(* CODESYS project WagoLibVisuIndustrialElements.library
   Description: Visualization objects for use with e!Cockpit programming environment
   Version: 1.0.0
   Title: WagoLibIndustrialVisuElements
   Author: JCox
   CompiledLibraryCompatibilityVersion: CODESYS V3.5 SP16 Patch 2
   Company: WAGO Corp. USA

Project tree, tasks and I/O mapping:
  libraries: VisuSymbols, 3.5.17.0 (System); WagoVisuIcons, 1.1.0.4 (WAGO)
  5ce3da45-db07-42e7-a21c-a00fff4ed8f6|Z:\Dropbox\Demos\Image Library\JPG Exports\blower1.png
  text list GlobalTextList
  5ce3da45-db07-42e7-a21c-a00fff4ed8f6|Z:\Dropbox\Demos\Image Library\JPG Exports\barrelblue.png
  visualisation GateValve1
  visualisation GlobeValve1
  visualisation Motor1
  visualisation Motor2
  visualisation Pump1
  visualisation Pump2
  visualisation Pump3
  visualisation Pump4
  visualisation Tank1
  visualisation Tank2
  visualisation Tank3
  visualisation Tank4
  visualisation Valve1
  visualisation Valve2
  image pool ImagePool
  5ce3da45-db07-42e7-a21c-a00fff4ed8f6|Z:\Dropbox\Demos\Image Library\JPG Exports\boiler1.png
  5ce3da45-db07-42e7-a21c-a00fff4ed8f6|Z:\Dropbox\Demos\Image Library\JPG Exports\barrelred.png
  visualisation Burner1
  5ce3da45-db07-42e7-a21c-a00fff4ed8f6|Z:\Dropbox\Demos\Image Library\JPG Exports\heatpipeOFF.png
  5ce3da45-db07-42e7-a21c-a00fff4ed8f6|Z:\Dropbox\Demos\Image Library\JPG Exports\heatpipeON.png
  5ce3da45-db07-42e7-a21c-a00fff4ed8f6|Z:\Dropbox\Demos\Image Library\JPG Exports\boiler2.png
  5ce3da45-db07-42e7-a21c-a00fff4ed8f6|Z:\Dropbox\Demos\Image Library\JPG Exports\box1.png
  5ce3da45-db07-42e7-a21c-a00fff4ed8f6|Z:\Dropbox\Demos\Image Library\JPG Exports\box2.png
  5ce3da45-db07-42e7-a21c-a00fff4ed8f6|Z:\Dropbox\Demos\Image Library\JPG Exports\check valveGRN.png
  5ce3da45-db07-42e7-a21c-a00fff4ed8f6|Z:\Dropbox\Demos\Image Library\JPG Exports\check valveGRN2.png
  5ce3da45-db07-42e7-a21c-a00fff4ed8f6|Z:\Dropbox\Demos\Image Library\JPG Exports\check valveGRY.png
  5ce3da45-db07-42e7-a21c-a00fff4ed8f6|Z:\Dropbox\Demos\Image Library\JPG Exports\check valveGRY2.png
  5ce3da45-db07-42e7-a21c-a00fff4ed8f6|Z:\Dropbox\Demos\Image Library\JPG Exports\check valveRED.png
  5ce3da45-db07-42e7-a21c-a00fff4ed8f6|Z:\Dropbox\Demos\Image Library\JPG Exports\check valveRED2.png
  5ce3da45-db07-42e7-a21c-a00fff4ed8f6|Z:\Dropbox\Demos\Image Library\JPG Exports\conveyor1.png
  5ce3da45-db07-42e7-a21c-a00fff4ed8f6|Z:\Dropbox\Demos\Image Library\JPG Exports\conveyor3.png
  5ce3da45-db07-42e7-a21c-a00fff4ed8f6|Z:\Dropbox\Demos\Image Library\JPG Exports\fireEMPTY.png
  5ce3da45-db07-42e7-a21c-a00fff4ed8f6|Z:\Dropbox\Demos\Image Library\JPG Exports\fireFULL.png
  5ce3da45-db07-42e7-a21c-a00fff4ed8f6|Z:\Dropbox\Demos\Image Library\JPG Exports\gatevalveGRN.png
  5ce3da45-db07-42e7-a21c-a00fff4ed8f6|Z:\Dropbox\Demos\Image Library\JPG Exports\gatevalveGRY.png
  5ce3da45-db07-42e7-a21c-a00fff4ed8f6|Z:\Dropbox\Demos\Image Library\JPG Exports\globevalveGRN.png
  5ce3da45-db07-42e7-a21c-a00fff4ed8f6|Z:\Dropbox\Demos\Image Library\JPG Exports\globevalveGRY.png
  5ce3da45-db07-42e7-a21c-a00fff4ed8f6|Z:\Dropbox\Demos\Image Library\JPG Exports\mixer1GRN.png
  5ce3da45-db07-42e7-a21c-a00fff4ed8f6|Z:\Dropbox\Demos\Image Library\JPG Exports\mixer1RED.png
  5ce3da45-db07-42e7-a21c-a00fff4ed8f6|Z:\Dropbox\Demos\Image Library\JPG Exports\motor1.png
  5ce3da45-db07-42e7-a21c-a00fff4ed8f6|Z:\Dropbox\Demos\Image Library\JPG Exports\motor1GRN.png
  5ce3da45-db07-42e7-a21c-a00fff4ed8f6|Z:\Dropbox\Demos\Image Library\JPG Exports\motor1RED.png
  5ce3da45-db07-42e7-a21c-a00fff4ed8f6|Z:\Dropbox\Demos\Image Library\JPG Exports\motorBLU1.png
  5ce3da45-db07-42e7-a21c-a00fff4ed8f6|Z:\Dropbox\Demos\Image Library\JPG Exports\motorBLU2.png
  5ce3da45-db07-42e7-a21c-a00fff4ed8f6|Z:\Dropbox\Demos\Image Library\JPG Exports\motorBLU3.png
  5ce3da45-db07-42e7-a21c-a00fff4ed8f6|Z:\Dropbox\Demos\Image Library\JPG Exports\motorGRN1.png
  5ce3da45-db07-42e7-a21c-a00fff4ed8f6|Z:\Dropbox\Demos\Image Library\JPG Exports\motorGRN2.png
  5ce3da45-db07-42e7-a21c-a00fff4ed8f6|Z:\Dropbox\Demos\Image Library\JPG Exports\motorGRN3.png
  5ce3da45-db07-42e7-a21c-a00fff4ed8f6|Z:\Dropbox\Demos\Image Library\JPG Exports\motorRED1.png
  5ce3da45-db07-42e7-a21c-a00fff4ed8f6|Z:\Dropbox\Demos\Image Library\JPG Exports\motorRED2.png
  5ce3da45-db07-42e7-a21c-a00fff4ed8f6|Z:\Dropbox\Demos\Image Library\JPG Exports\motorRED3.png
  5ce3da45-db07-42e7-a21c-a00fff4ed8f6|Z:\Dropbox\Demos\Image Library\JPG Exports\pipe1H.png
  5ce3da45-db07-42e7-a21c-a00fff4ed8f6|Z:\Dropbox\Demos\Image Library\JPG Exports\pipe1V.png
  5ce3da45-db07-42e7-a21c-a00fff4ed8f6|Z:\Dropbox\Demos\Image Library\JPG Exports\pipeJ1.png
  5ce3da45-db07-42e7-a21c-a00fff4ed8f6|Z:\Dropbox\Demos\Image Library\JPG Exports\pipeJ2.png
  5ce3da45-db07-42e7-a21c-a00fff4ed8f6|Z:\Dropbox\Demos\Image Library\JPG Exports\pipeJ3.png
  5ce3da45-db07-42e7-a21c-a00fff4ed8f6|Z:\Dropbox\Demos\Image Library\JPG Exports\pipeJ4.png
  5ce3da45-db07-42e7-a21c-a00fff4ed8f6|Z:\Dropbox\Demos\Image Library\JPG Exports\pipeT1.png
  5ce3da45-db07-42e7-a21c-a00fff4ed8f6|Z:\Dropbox\Demos\Image Library\JPG Exports\pipeT2.png
  5ce3da45-db07-42e7-a21c-a00fff4ed8f6|Z:\Dropbox\Demos\Image Library\JPG Exports\pipeT3.png
  5ce3da45-db07-42e7-a21c-a00fff4ed8f6|Z:\Dropbox\Demos\Image Library\JPG Exports\pipeT4.png
  5ce3da45-db07-42e7-a21c-a00fff4ed8f6|Z:\Dropbox\Demos\Image Library\JPG Exports\pipeX.png
  5ce3da45-db07-42e7-a21c-a00fff4ed8f6|Z:\Dropbox\Demos\Image Library\JPG Exports\pump1.png
  5ce3da45-db07-42e7-a21c-a00fff4ed8f6|Z:\Dropbox\Demos\Image Library\JPG Exports\pump2.png
  5ce3da45-db07-42e7-a21c-a00fff4ed8f6|Z:\Dropbox\Demos\Image Library\JPG Exports\pump3.png
  5ce3da45-db07-42e7-a21c-a00fff4ed8f6|Z:\Dropbox\Demos\Image Library\JPG Exports\pump4.png
  5ce3da45-db07-42e7-a21c-a00fff4ed8f6|Z:\Dropbox\Demos\Image Library\JPG Exports\tank2.png
  5ce3da45-db07-42e7-a21c-a00fff4ed8f6|Z:\Dropbox\Demos\Image Library\JPG Exports\tank1.png
  5ce3da45-db07-42e7-a21c-a00fff4ed8f6|Z:\Dropbox\Demos\Image Library\JPG Exports\tank3.png
  5ce3da45-db07-42e7-a21c-a00fff4ed8f6|Z:\Dropbox\Demos\Image Library\JPG Exports\tank4.png
  5ce3da45-db07-42e7-a21c-a00fff4ed8f6|Z:\Dropbox\Demos\Image Library\JPG Exports\tank5.png
  5ce3da45-db07-42e7-a21c-a00fff4ed8f6|Z:\Dropbox\Demos\Image Library\JPG Exports\tank6.png
  5ce3da45-db07-42e7-a21c-a00fff4ed8f6|Z:\Dropbox\Demos\Image Library\JPG Exports\tank7.png
*)

// /GateValve1
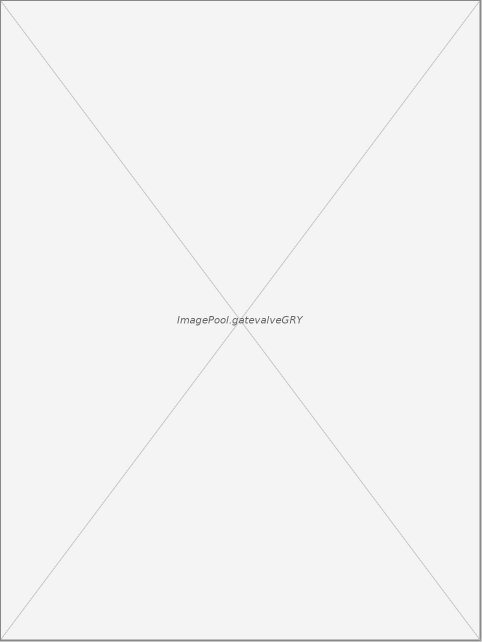
VISUALIZATION GateValve1  // 482x642
VAR_IN_OUT
	xOn		: BOOL;
END_VAR
    Image (0,0 480x640), invisible if: NOT xOn, image: ImagePool.gatevalveGRN
    Image (0,0 480x640), invisible if: xOn, image: ImagePool.gatevalveGRY
END_VISUALIZATION

// /GlobeValve1
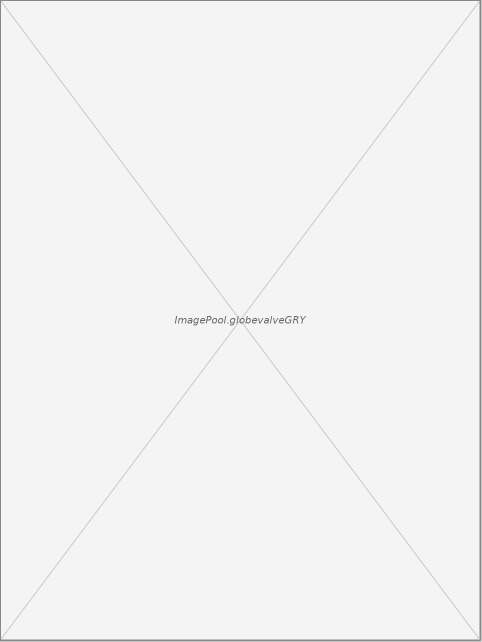
VISUALIZATION GlobeValve1  // 482x642
VAR_IN_OUT
	xOn		: BOOL;
END_VAR
    Image (0,0 480x640), invisible if: NOT xOn, image: ImagePool.globevalveGRN
    Image (0,0 480x640), invisible if: xOn, image: ImagePool.globevalveGRY
END_VISUALIZATION

// /Motor1
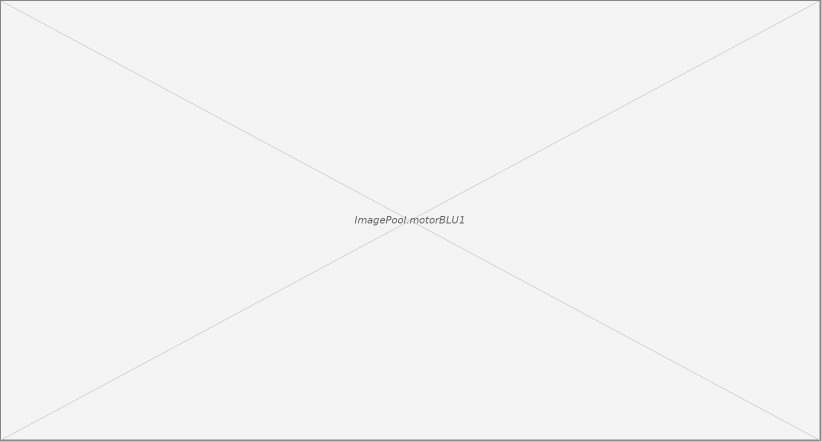
VISUALIZATION Motor1  // 822x442
VAR_IN_OUT
	xOn	: BOOL;
END_VAR
    Image (0,0 820x440), invisible if: NOT xOn, image: ImagePool.motorGRN1
    Image (0,0 820x440), invisible if: xOn, image: ImagePool.motorBLU1
END_VISUALIZATION

// /Motor2
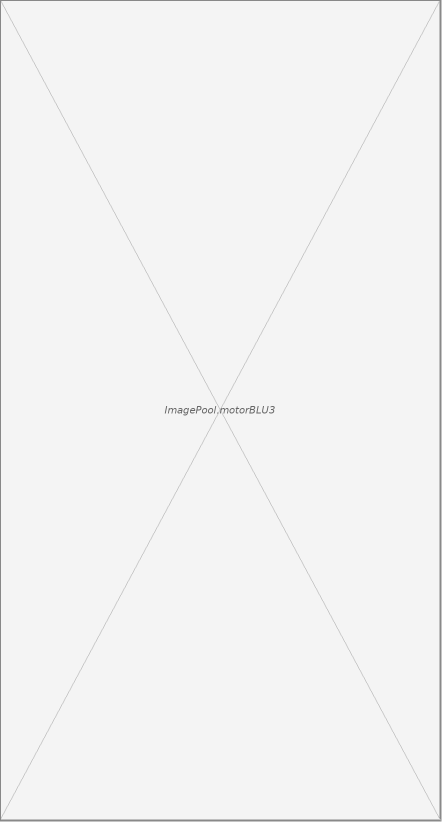
VISUALIZATION Motor2  // 442x822
VAR_IN_OUT
	xOn	: BOOL;
END_VAR
    Image (0,0 440x820), invisible if: NOT xOn, image: ImagePool.motorGRN3
    Image (0,0 440x820), invisible if: xOn, image: ImagePool.motorBLU3
END_VISUALIZATION

// /Pump1
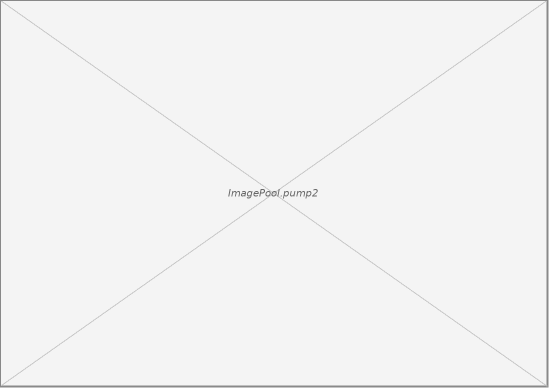
VISUALIZATION Pump1  // 549x388
VAR_IN_OUT
	xGo	: BOOL;
END_VAR
    Ellipse (125,44 300x300), colour toggle: xGo
    Image (0,0 547x386), image: ImagePool.pump2
END_VISUALIZATION

// /Pump2
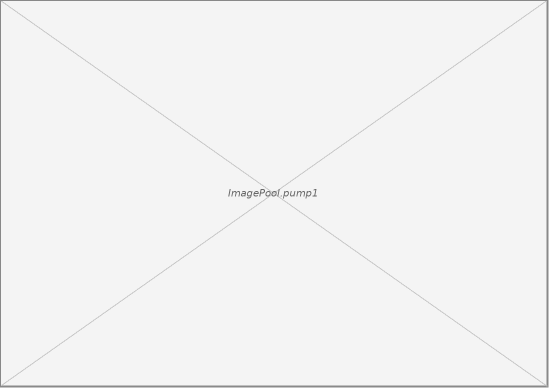
VISUALIZATION Pump2  // 549x388
VAR_IN_OUT
	xGo	: BOOL;
END_VAR
    Ellipse (125,44 300x300), colour toggle: xGo
    Image (0,0 547x386), image: ImagePool.pump1
END_VISUALIZATION

// /Pump3
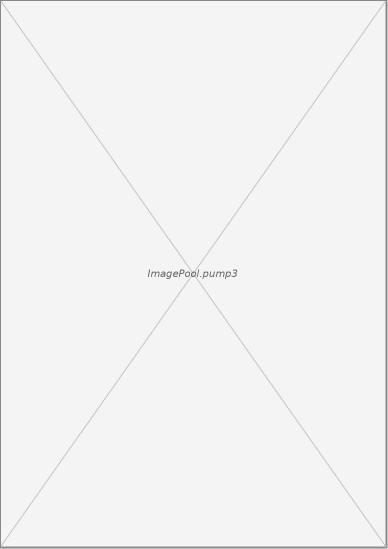
VISUALIZATION Pump3  // 388x549
VAR_IN_OUT
	xGo	: BOOL;
END_VAR
    Ellipse (47,122 300x300), colour toggle: xGo
    Image (0,0 386x547), image: ImagePool.pump3
END_VISUALIZATION

// /Pump4
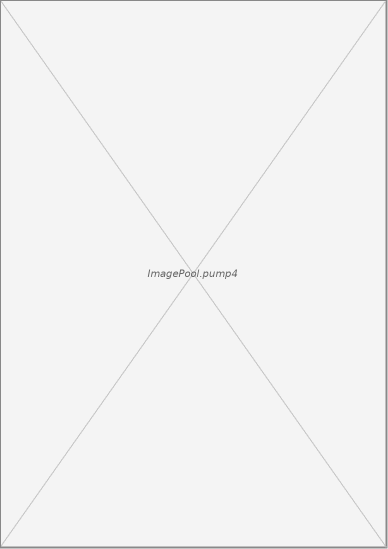
VISUALIZATION Pump4  // 388x549
VAR_IN_OUT
	xGo	: BOOL;
END_VAR
    Ellipse (47,122 300x300), colour toggle: xGo
    Image (0,0 386x547), image: ImagePool.pump4
END_VISUALIZATION

// /Tank1
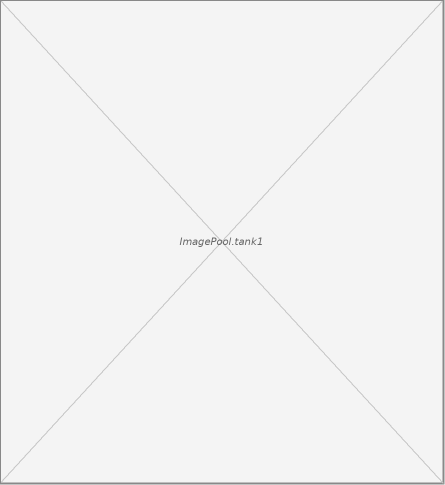
VISUALIZATION Tank1  // 445x485
VAR_IN_OUT
	diBar		: DINT;
END_VAR
    BarDisplayImage (35,38 65x410), value: diBar, style: BarDisplayImage-Gray, scale format: %.1f, scale 0..1000
    Image (0,0 443x483), image: ImagePool.tank1
END_VISUALIZATION

// /Tank2
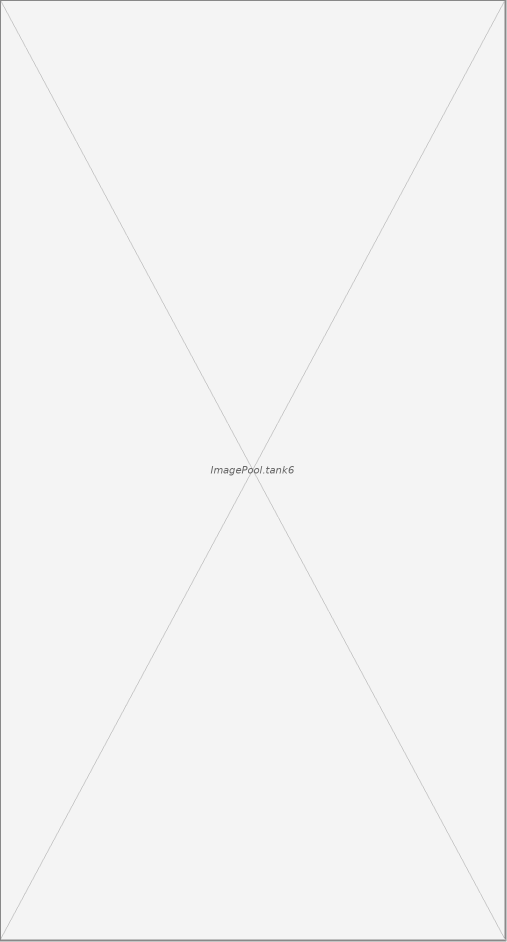
VISUALIZATION Tank2  // 507x942
VAR_IN_OUT
	diBar		: DINT;
END_VAR
    BarDisplayImage (45,131 65x777), value: diBar, style: BarDisplayImage-Gray, scale format: %.1f, scale 0..1000
    Image (0,0 505x940), image: ImagePool.tank6
END_VISUALIZATION

// /Tank3
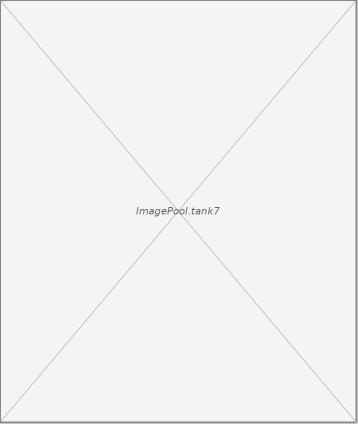
VISUALIZATION Tank3  // 358x424
VAR_IN_OUT
	diBar		: DINT;
END_VAR
    BarDisplayImage (189,21 78x306), value: diBar, style: BarDisplayImage-Gray, scale format: %.1f, scale 0..1000
    Image (0,0 356x422), image: ImagePool.tank7
END_VISUALIZATION

// /Tank4
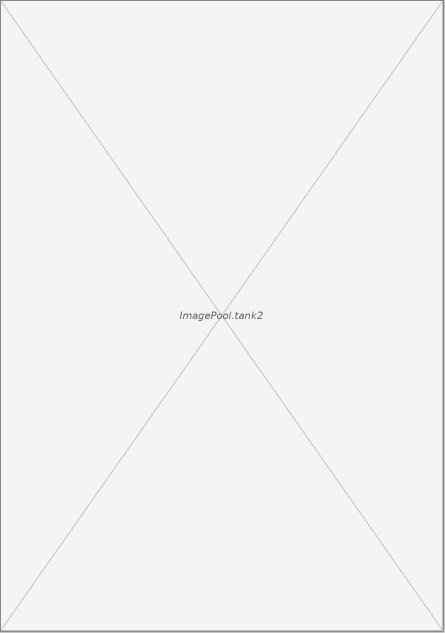
VISUALIZATION Tank4  // 445x633
VAR_IN_OUT
	diBar		: DINT;
END_VAR
    BarDisplayImage (33,118 65x471), value: diBar, style: BarDisplayImage-Gray, scale format: %.1f, scale 0..1000
    Image (0,0 443x631), image: ImagePool.tank2
END_VISUALIZATION

// /Valve1
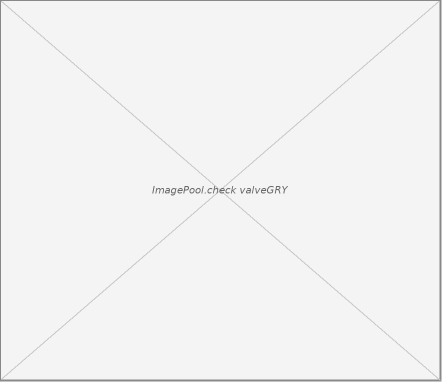
VISUALIZATION Valve1  // 442x382
VAR_IN_OUT
	xOn		: BOOL;
END_VAR
    Image (0,0 440x380), invisible if: NOT xOn, image: ImagePool.check valveGRN
    Image (0,0 440x380), invisible if: xOn, image: ImagePool.check valveGRY
END_VISUALIZATION

// /Valve2
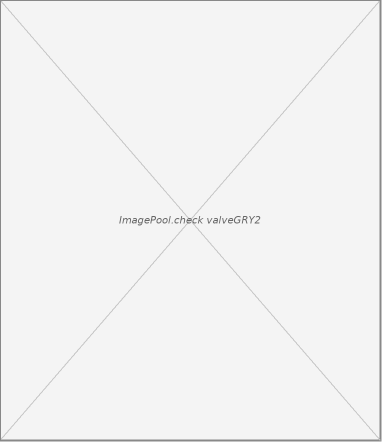
VISUALIZATION Valve2  // 382x442
VAR_IN_OUT
	xOn		: BOOL;
END_VAR
    Image (0,0 380x440), invisible if: NOT xOn, image: ImagePool.check valveGRN2
    Image (0,0 380x440), invisible if: xOn, image: ImagePool.check valveGRY2
END_VISUALIZATION

// /Burner1
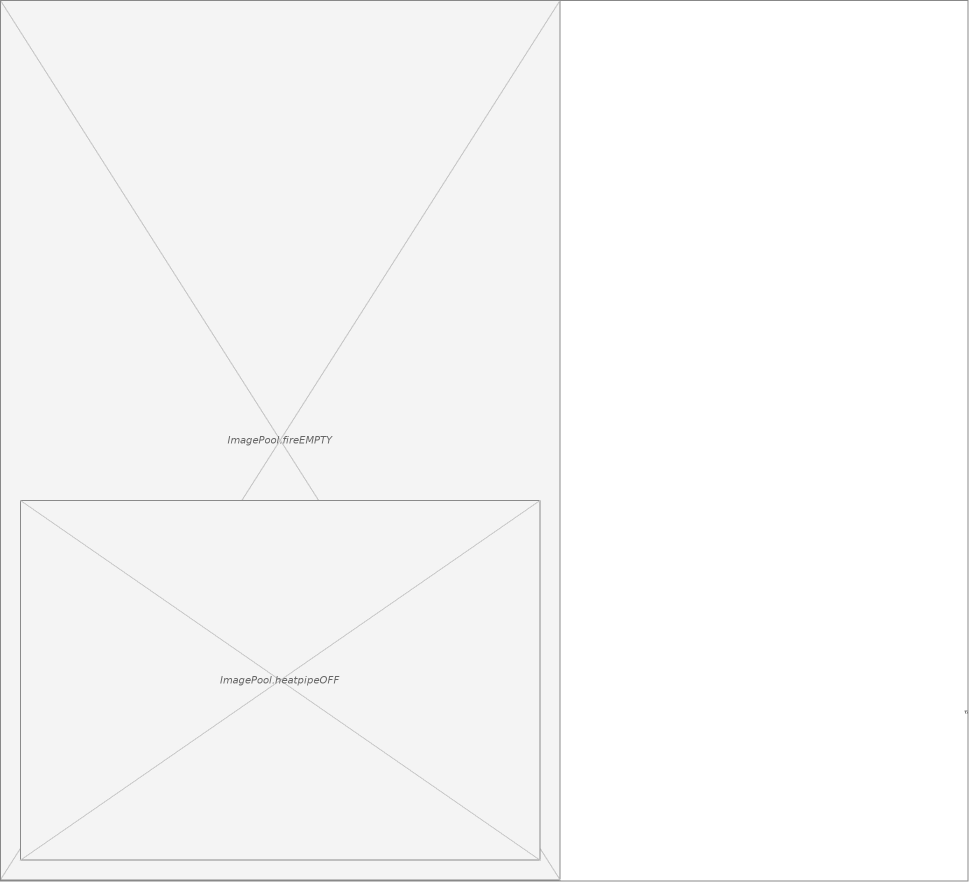
VISUALIZATION Burner1  // 969x882
VAR_IN_OUT
	xOn		: BOOL;
END_VAR
    Image (20,500 520x360), invisible if: NOT xOn, image: ImagePool.heatpipeON
    Image (0,0 560x880), image: ImagePool.fireEMPTY
    Image (20,500 520x360), invisible if: xOn, image: ImagePool.heatpipeOFF
    Button (967,712 0x1)
END_VISUALIZATION
